(* CODESYS project Tc2_AiSampleLib.library
   Company: Beckhoff Automation
   Version: 1.0.0.0
   Title: Tc2_AiSampleLib

Project tree, tasks and I/O mapping:
  libraries: Tc2_Standard, * (Beckhoff Automation GmbH); Tc2_System, * (Beckhoff Automation GmbH); Tc3_Interfaces, * (Beckhoff Automation GmbH); Tc3_Module, * (Beckhoff Automation GmbH)
  DUTs/
  GVLs/
  POUs/
    function block FB_SamplePou [ST]
    program MAIN [ST]
  Version/
    global variables Global_Version
  VISUs/
*)

// Version/Global_Version
// This function has been automatically generated from the project information.
VAR_GLOBAL CONSTANT
	{attribute 'const_non_replaced'}
	stLibVersion_Tc2_AiSampleLib : ST_LibVersion := (iMajor := 1, iMinor := 0, iBuild := 0, iRevision := 0, sVersion := '1.0.0.0');
END_VAR

// POUs/FB_SamplePou
FUNCTION_BLOCK FB_SamplePou
VAR_INPUT
	bInput	:	BOOL;
END_VAR
VAR_OUTPUT
	bOuput	:	BOOL;
END_VAR
VAR
END_VAR

bOutput := bInput;

END_FUNCTION_BLOCK

// POUs/MAIN
PROGRAM MAIN
VAR
END_VAR

END_PROGRAM
